(* CODESYS project AICodesAndValidation.library
   LanguageModelAttribute: qualified-access-only
   Author: Wiktor Pytka
   Version: 1.0.0.0
   Title: AI Codes And Validation
   Placeholder: CODE
   DefaultNamespace: CODE
   Company: Marden Edwards

Project tree, tasks and I/O mapping:
  libraries: Tc2_Standard, * (Beckhoff Automation GmbH); Tc2_System, * (Beckhoff Automation GmbH)
  DUTs/
    AI Codes And Validation/
      data type E_CodeAI
      data type E_CodeType
      data type ST_CodeInfo
      data type ST_CodeValidation
  GVLs/
  POUs/
    AI Codes And Validation FBs/
      function F_AssignValToStringWithPrefix [ST]
      function F_GetItemAI [ST]
      function block FB_ClearCodeInfo [ST]
      function block FB_ValidateExplicitCode [ST]
  Version/
    global variables Global_Version
  VISUs/
*)

// DUTs/AI Codes And Validation/E_CodeAI
{attribute 'qualified_only'}
TYPE E_CodeAI :
(
	GTIN 			:= 1,
	BATCH 			:= 10,
	SERIAL			:= 21,
	PO				:= 91,
	BRANDSPEC		:= 92,
	CRYPTO			:= 93,
	PRODDATE		:= 94,
	RSKU 			:= 240,
	MRP				:= 8005,
	USERFIELD		:= 999
);
END_TYPE

// DUTs/AI Codes And Validation/E_CodeType
TYPE E_CodeType :
(
	E_NONE,
	E_PACK,
	E_INTERIM,
	E_OUTER,
	E_CASE

);
END_TYPE

// DUTs/AI Codes And Validation/ST_CodeInfo
TYPE ST_CodeInfo :
STRUCT
	eCodeType					:	E_CodeType;

	nMinLength					: 	INT;
	nEntireLength				:	INT;
	bValidateEntireLength		: 	BOOL;
	nNumberOfAIs				:	INT;

	stGTIN 						:	ST_CodeValidation	:=		(sFieldName :='GTIN',					bNameEditable := FALSE, 		nGS1_AI := 1);
	stBatchID 					:	ST_CodeValidation	:=		(sFieldName :='BatchID', 				bNameEditable := FALSE, 		nGS1_AI := 10);
	stSerialCode 				:	ST_CodeValidation	:=		(sFieldName :='SerialCode', 			bNameEditable := FALSE, 		nGS1_AI := 21);
	stProductionOrder 			:	ST_CodeValidation	:=		(sFieldName :='ProductionOrder', 		bNameEditable := FALSE, 		nGS1_AI := 91);
	stCryptoCode				:	ST_CodeValidation	:=		(sFieldName :='CryptoCode', 			bNameEditable := FALSE, 		nGS1_AI := 93);
	stRSKU						:	ST_CodeValidation	:=		(sFieldName :='RSKU', 					bNameEditable := FALSE, 		nGS1_AI := 240);
	stMRP		 				:	ST_CodeValidation	:=		(sFieldName :='MRP', 					bNameEditable := FALSE, 		nGS1_AI := 8005);
	stBrandSpecification		:	ST_CodeValidation	:=		(sFieldName :='BrandSpec',				bNameEditable := FALSE, 		nGS1_AI := 92);
	stProduceDate				:	ST_CodeValidation	:=		(sFieldName :='ProduceDate',			bNameEditable := TRUE, 			nGS1_AI := 94);
	stUserField3				:	ST_CodeValidation	:=		(sFieldName :='',						bNameEditable := TRUE, 			nGS1_AI := 95);

END_STRUCT
END_TYPE

// DUTs/AI Codes And Validation/ST_CodeValidation
TYPE ST_CodeValidation :
STRUCT
	bValidate 			:	BOOL;

	sFieldName		:	STRING(15)	:='';
	bNameEditable	:	BOOL;
	nListPosition		: 	BYTE;

	sStartAI 			: 	STRING(6)		:= '';
	sEndAI 			: 	STRING(6) 	:= '';
	nCodeStartPos		:	INT;
	nCodeLength		:	INT;

	nGS1_AI			: 	INT;

(* If sStartAI is empty, then use nCodeStartPos, else find sStartAI in code for start position *)
(* If sEndAI is empty then use nCodeLength, else find sEndAI in code for end position*)

(*General Application Idendifiers (AI) Description:
	01:		GTIN
	10: 		Batch ID
	21: 		Serial Code
	91:		Production Order
	93:		Crypto
	240:		RSKU
*)

END_STRUCT
END_TYPE

// Version/Global_Version
{attribute 'TcGenerated'}
{attribute 'no-analysis'}
{attribute 'linkalways'}
// This function has been automatically generated from the project information.
VAR_GLOBAL CONSTANT
	{attribute 'const_non_replaced'}
	stLibVersion_AI_Codes_And_Validation : ST_LibVersion := (iMajor := 1, iMinor := 0, iBuild := 0, iRevision := 0, sVersion := '1.0.0.0');
END_VAR

// POUs/AI Codes And Validation FBs/F_AssignValToStringWithPrefix
FUNCTION F_AssignValToStringWithPrefix : T_MaxString
VAR_INPUT
	asRejectReason		: T_MaxString;
	anValue				: ARRAY[0..10] OF STRING(10);
	asPointer          	  		: ARRAY[0..10] OF STRING(10);
	nPrefixSize			: UINT;
	nPrefixValue			: STRING(5);
END_VAR

VAR
	(*bPointerNotFound	           : BOOL;*)
	nCounter				: INT;
	nPointerPos			: INT;
	asAssignedRejectReason	: T_MaxString;
	sValToAssign			: STRING(20);
END_VAR

(* This Function assigns value to predefined Pointer in string.
     Function can assing up to 10 Values
     For ex. string Reject Reason := 'XXDUPn1-n2XX'
     	         nValue := [3, 4], sPointer := ['n1', 'n2']		
	         asRejectReason := 'XXDUP3-4XX'	*)

F_AssignValToStringWithPrefix := '';

asAssignedRejectReason := asRejectReason;

REPEAT
	nPointerPos := FIND(asAssignedRejectReason, asPointer[nCounter]);
	IF nPointerPos > 0 AND  asPointer[nCounter] <> '' THEN
		sValToAssign :=  F_StringAddPrefix(anValue[nCounter], nPrefixSize, nPrefixValue);
		 asAssignedRejectReason := REPLACE(asAssignedRejectReason, sValToAssign, LEN(asPointer[nCounter]), nPointerPos);
	END_IF;
	nCounter := nCounter + 1;
UNTIL
	nCounter >= 10
END_REPEAT

IF nCounter <> 0 THEN
	F_AssignValToStringWithPrefix := asAssignedRejectReason;
ELSE
	F_AssignValToStringWithPrefix := asRejectReason;
END_IF;

END_FUNCTION

// POUs/AI Codes And Validation FBs/F_GetItemAI
FUNCTION F_GetItemAI : T_MaxString
VAR_INPUT
	sFullCode		: T_MaxString;
	eCodeType		: E_CodeAI;
	stCodeInfo		: ST_CodeInfo;
END_VAR
VAR
	stItem			: ST_CodeValidation;
	
	sTemp			: T_MaxString;
	nStart			: INT;
	nEnd			: INT;
	
	sResultString	: T_MaxString;
END_VAR

IF stCodeInfo.nEntireLength > 0 THEN

	IF eCodeType = E_CodeAI.GTIN THEN 			stItem := stCodeInfo.stGTIN;
	ELSIF eCodeType = E_CodeAI.BATCH THEN 		stItem := stCodeInfo.stBatchID;
	ELSIF eCodeType = E_CodeAI.SERIAL THEN		stItem := stCodeInfo.stSerialCode;
	ELSIF eCodeType = E_CodeAI.PO THEN			stItem := stCodeInfo.stProductionOrder;
	ELSIF eCodeType = E_CodeAI.CRYPTO THEN		stItem := stCodeInfo.stCryptoCode;
	ELSIF eCodeType = E_CodeAI.RSKU THEN		stItem := stCodeInfo.stRSKU;
	ELSIF eCodeType = E_CodeAI.MRP THEN			stItem := stCodeInfo.stMRP;
	ELSIF eCodeType = E_CodeAI.BRANDSPEC THEN	stItem := stCodeInfo.stBrandSpecification;
	ELSIF eCodeType = E_CodeAI.PRODDATE THEN	stItem := stCodeInfo.stProduceDate;
	ELSIF eCodeType = E_CodeAI.USERFIELD THEN	stItem := stCodeInfo.stUserField3;
	END_IF

/////////////////////////////////////////////////////////////////////////////////////////////////////

	IF stItem.sStartAI <> '' AND stItem.sEndAI <> '' THEN
		
		nStart := FIND(sFullCode, stItem.sStartAI) + LEN(stItem.sStartAI);
		
		IF nStart > 0 THEN
			sTemp := RIGHT(sFullCode, LEN(sFullCode) - (nStart - 1));
		ELSE
			sTemp := sFullCode;
		END_IF
		
		nEnd := FIND(sTemp, stItem.sEndAI);
		
		IF nEnd = 0 THEN
			nEnd := LEN(sFullCode)+1;
		ELSE
			nEnd := nEnd +(nStart - 1);
		END_IF
		
	ELSIF stItem.sStartAI <> '' AND stItem.nCodeLength > 0 THEN
		
		nStart := FIND(sFullCode, stItem.sStartAI) + LEN(stItem.sStartAI);
		nEnd := nStart + stItem.nCodeLength;
		
	ELSIF stItem.nCodeStartPos > 0 AND stItem.sEndAI <> '' THEN
		
		nStart := stItem.nCodeStartPos;
		sTemp := RIGHT(sFullCode, LEN(sFullCode) - (nStart - 1));
		nEnd := FIND(sTemp, stItem.sEndAI);
		
		IF nEnd = 0 THEN
			nEnd := LEN(sFullCode)+1;
		ELSE
			nEnd := nEnd +(nStart - 1);
		END_IF
		
	ELSIF stItem.nCodeStartPos >= 0 AND stItem.nCodeLength > 0 THEN
		
		nStart := stItem.nCodeStartPos;
		nEnd := nStart + stItem.nCodeLength;
	ELSE
		nStart := 0;
		nEnd := 0;
	END_IF
	
	IF nStart > 0 AND nEnd > 0 THEN
		sResultString := MID(sFullCode, nEnd - nStart, nStart);
	ELSE
		sResultString := '';
	END_IF
ELSE
	sResultString := '';
END_IF

F_GetItemAI := sResultString;

END_FUNCTION

// POUs/AI Codes And Validation FBs/FB_ClearCodeInfo
FUNCTION_BLOCK FB_ClearCodeInfo
VAR_INPUT
END_VAR
VAR_IN_OUT
	stCodeInfo						: ST_CodeInfo;
END_VAR
VAR
	sMemoUserField					: STRING;
END_VAR

IF stCodeInfo.stGTIN.nListPosition = 0 THEN
	MEMSET(ADR(stCodeInfo.stGTIN), 16#00, SIZEOF(stCodeInfo.stGTIN));
	stCodeInfo.stGTIN.sFieldName :='GTIN';
	stCodeInfo.stGTIN.nGS1_AI := 1;
END_IF
IF stCodeInfo.stBatchID.nListPosition  = 0 THEN
	MEMSET(ADR(stCodeInfo.stBatchID), 16#00, SIZEOF(stCodeInfo.stBatchID));
	stCodeInfo.stBatchID.sFieldName :='BatchID';
	stCodeInfo.stBatchID.nGS1_AI := 10;
END_IF
IF stCodeInfo.stSerialCode.nListPosition = 0 THEN
	MEMSET(ADR(stCodeInfo.stSerialCode), 16#00, SIZEOF(stCodeInfo.stSerialCode));
	stCodeInfo.stSerialCode.sFieldName :='SerialCode';
	stCodeInfo.stSerialCode.nGS1_AI := 21;
END_IF
IF stCodeInfo.stProductionOrder.nListPosition  = 0 THEN
	MEMSET(ADR(stCodeInfo.stProductionOrder), 16#00, SIZEOF(stCodeInfo.stProductionOrder));
	stCodeInfo.stProductionOrder.sFieldName :='ProductionOrder';
	stCodeInfo.stProductionOrder.nGS1_AI := 91;
END_IF
IF stCodeInfo.stCryptoCode.nListPosition = 0 THEN
	MEMSET(ADR(stCodeInfo.stCryptoCode), 16#00, SIZEOF(stCodeInfo.stCryptoCode));
	stCodeInfo.stCryptoCode.sFieldName :='CryptoCode';
	stCodeInfo.stCryptoCode.nGS1_AI := 93;
END_IF
IF stCodeInfo.stRSKU.nListPosition = 0 THEN
	MEMSET(ADR(stCodeInfo.stRSKU), 16#00, SIZEOF(stCodeInfo.stRSKU));
	stCodeInfo.stRSKU.sFieldName :='SKU';
	stCodeInfo.stRSKU.nGS1_AI := 240;
END_IF
IF stCodeInfo.stMRP.nListPosition = 0 THEN
	MEMSET(ADR(stCodeInfo.stMRP), 16#00, SIZEOF(stCodeInfo.stMRP));
	stCodeInfo.stMRP.sFieldName :='MRP';
	stCodeInfo.stMRP.nGS1_AI := 8005;
END_IF
IF stCodeInfo.stBrandSpecification.nListPosition = 0 THEN
	MEMSET(ADR(stCodeInfo.stBrandSpecification), 16#00, SIZEOF(stCodeInfo.stBrandSpecification));
	stCodeInfo.stBrandSpecification.sFieldName := 'BrandSpec';
	stCodeInfo.stBrandSpecification.nGS1_AI := 92;
END_IF
IF stCodeInfo.stProduceDate.nListPosition = 0 THEN
	MEMSET(ADR(stCodeInfo.stProduceDate), 16#00, SIZEOF(stCodeInfo.stProduceDate));
	stCodeInfo.stProduceDate.sFieldName :='ProduceDate';
	stCodeInfo.stProduceDate.nGS1_AI := 94;
END_IF
IF stCodeInfo.stUserField3.nListPosition  = 0THEN
	sMemoUserField := stCodeInfo.stUserField3.sFieldName;
	MEMSET(ADR(stCodeInfo.stUserField3), 16#00, SIZEOF(stCodeInfo.stUserField3));
	stCodeInfo.stUserField3.sFieldName :=sMemoUserField;
	stCodeInfo.stUserField3.nGS1_AI := 95;
END_IF

END_FUNCTION_BLOCK

// POUs/AI Codes And Validation FBs/FB_ValidateExplicitCode
FUNCTION_BLOCK FB_ValidateExplicitCode
VAR_INPUT
	sFullCode					: STRING(255);
	stCodeInfo				: ST_CodeInfo;
	stProductInstruction			: ST_PCM_Status;
END_VAR
VAR_OUTPUT
	bValidationOK				: BOOL;
	bEntireCodeLengthOK		: BOOL;

	bGtinOK					: BOOL;
	bSerialCodeOK				: BOOL;
	bBatchIDOK				: BOOL;
	bProductionOrderOK		: BOOL;
	bCryptoOK				: BOOL;
	bRskuOK					: BOOL;
	bMRPOK					: BOOL;
	bBrandOK				: BOOL;
	bProduceDateOK		: BOOL;

	sGTIN					: T_CodeGTIN;
	sSerial					: STRING(255);
	sBatchID					: T_CodeBATCH;
	sProductionOrder			: T_CodePO;
	sCrypto					: STRING(20);
	sRSKU					: T_CodeRSKU;
	sMRP					: STRING(8);
	sBrand					: T_CodeBRAND;
	sProduceDate			: T_CodePRODUCEDATE;

END_VAR
VAR
	eCodeAIType					: E_CodeAIType;
	sGtinToValidateAgainst		: T_CodeGTIN;
	sBrandToValidateAgainst		: T_CodeBRAND;
END_VAR

(***********************************************
	GTIN 			= 1;
	BatchID 			= 10;
	SerialCode		= 21;
	ProductionOrder 	= 91;
	CryptoCode		= 93;
	RSKU 			= 240;
	MRP				= 8005;
	BrandSpecification = 92
	ProduceDate		= 94
	UserField3

***********************************************)
(*
WHILE FIND(sFullCode, '$1D') > 0 DO
	sFullCode := DELETE(sFullCode, LEN('$1D'), FIND(sFullCode, '$1D'));
END_WHILE*)

sFullCode := F_ReplaceSingleChar(sFullCode, '$1D', '');

bEntireCodeLengthOK := (LEN(sFullCode) = stCodeInfo.nEntireLength) OR NOT(stCodeInfo.bValidateEntireLength);

CASE stCodeInfo.eCodeType OF

	E_PACK:
		sGtinToValidateAgainst := stProductInstruction.sPackGTIN;
		sBrandToValidateAgainst := LEFT(stProductInstruction.sPackBrandSpec, stCodeInfo.stBrandSpecification.nCodeLength);
	E_OUTER:
		sGtinToValidateAgainst := stProductInstruction.sOuterGTIN;
		sBrandToValidateAgainst := LEFT(stProductInstruction.sOuterBrandSpec, stCodeInfo.stBrandSpecification.nCodeLength);
	E_CASE:
		sGtinToValidateAgainst := stProductInstruction.sCaseGTIN;
		sBrandToValidateAgainst := LEFT(stProductInstruction.sCaseBrandSpec, stCodeInfo.stBrandSpecification.nCodeLength);
ELSE
		sGtinToValidateAgainst := '';
		sBrandToValidateAgainst := '';
END_CASE

sGTIN:= '';
sBatchID := '';
sSerial := '';
sProductionOrder := '';
sCrypto :='';
sRSKU := '';
sMRP :='';
sBrand := '';
sProduceDate :='';

bGtinOK := TRUE;
sGTIN := F_CODE_GetItem(sFullCode, eCodeAIType.GTIN, stCodeInfo);

IF stCodeInfo.stGTIN.bValidate THEN

	IF LEN(sGTIN) <> stCodeInfo.stGTIN.nCodeLength 	 OR
		 sGTIN <> sGtinToValidateAgainst 			THEN

		bGtinOK := FALSE;
	END_IF

END_IF

bBatchIDOK := TRUE;
sBatchID := F_CODE_GetItem(sFullCode, eCodeAIType.BatchID, stCodeInfo);

IF stCodeInfo.stBatchID.bValidate THEN

	IF LEN(sBatchID) <> stCodeInfo.stBatchID.nCodeLength 		 OR
		 sBatchID <> stProductInstruction.sBatchNumber		THEN

		bBatchIDOK := FALSE;
	END_IF

END_IF

bSerialCodeOK := TRUE;
sSerial := F_CODE_GetItem(sFullCode, eCodeAIType.SerialCode, stCodeInfo);

IF stCodeInfo.stSerialCode.bValidate AND stCodeInfo.stSerialCode.nCodeLength <> 0 THEN

	IF LEN(sSerial) <> stCodeInfo.stSerialCode.nCodeLength THEN
		bSerialCodeOK := FALSE;
	END_IF

END_IF

bProductionOrderOK := TRUE;
sProductionOrder := F_CODE_GetItem(sFullCode, eCodeAIType.ProductionOrder, stCodeInfo);

IF stCodeInfo.stProductionOrder.bValidate  THEN

	IF LEN(sProductionOrder) <> stCodeInfo.stProductionOrder.nCodeLength OR
		 sProductionOrder <> stProductInstruction.sProductionOrder	THEN

		bProductionOrderOK := FALSE;
	END_IF

END_IF

bCryptoOK := TRUE;
sCrypto := F_CODE_GetItem(sFullCode, eCodeAIType.CryptoCode, stCodeInfo);

IF stCodeInfo.stCryptoCode.bValidate AND stCodeInfo.stCryptoCode.nCodeLength <> 0 THEN

	IF LEN(sCrypto) <> stCodeInfo.stCryptoCode.nCodeLength THEN
		bCryptoOK := FALSE;
	END_IF

END_IF

bRskuOK := TRUE;
sRSKU := F_CODE_GetItem(sFullCode, eCodeAIType.RSKU, stCodeInfo);

IF stCodeInfo.stRSKU.bValidate THEN

	(*IF LEN(sRSKU) <> stCodeInfo.stRSKU.nCodeLength 	 OR
		 sRSKU <> stProductInstruction.sRetailSKU	THEN*)
	IF LEN(sRSKU) <> stCodeInfo.stRSKU.nCodeLength 	 OR
		( LEN(sRSKU) = 7 AND	stProductInstruction.sRetailSKU <> F_CASE_GetSKUFromHex(sRSKU)) 	OR
		( LEN(sRSKU) > 7 AND stProductInstruction.sRetailSKU <>  sRSKU) 	THEN

		bRskuOK := FALSE;
	END_IF

END_IF

bMRPOK := TRUE;
sMRP := F_CODE_GetItem(sFullCode, eCodeAIType.MRP, stCodeInfo);

IF stCodeInfo.stMRP.bValidate AND stCodeInfo.stMRP.nCodeLength <> 0 THEN

	IF LEN(sMRP) <> stCodeInfo.stMRP.nCodeLength THEN
		bMRPOK := FALSE;
	END_IF

END_IF

bBrandOK := TRUE;
sBrand := F_CODE_GetItem(sFullCode, eCodeAIType.BrandSpecification, stCodeInfo);

IF stCodeInfo.stBrandSpecification.bValidate THEN

	IF LEN(sBrand) <> stCodeInfo.stBrandSpecification.nCodeLength 	 OR
		 sBrand <> sBrandToValidateAgainst 			THEN

		bBrandOK := FALSE;
	END_IF

END_IF

bProduceDateOK := TRUE;
sProduceDate := F_CODE_GetItem(sFullCode, eCodeAIType.ProduceDate, stCodeInfo);

IF stCodeInfo.stProduceDate.bValidate AND stCodeInfo.stProduceDate.nCodeLength <> 0 THEN

	IF LEN(sProduceDate) <> stCodeInfo.stProduceDate.nCodeLength THEN
		bProduceDateOK := FALSE;
	END_IF

END_IF

bValidationOK := bGtinOK AND bBatchIDOK AND bSerialCodeOK  AND bProductionOrderOK AND bCryptoOK AND bRskuOK AND bMRPOK AND bBrandOK AND bProduceDateOK AND bEntireCodeLengthOK;

END_FUNCTION_BLOCK
